FUNCTION Call_HMI

hmiHeaderInstance(NameApplication := 'Hochregallager',
				  OperatingModeHMIInterface := hmiOperatingmodeInterface,
				  HeaderHMIInterface := hmiHeaderInterface);
			  
hmiAdsCommunicationInterfaceInstance(Timeout := T#1S,
									 TimeoutHMI := T#500ms,
									 LocalAdsPort := 851,
									 HeartbeatHMI := hmiAdsCommunicationInterface.HeartbeatHMI);
									 

hmiAdsCommunicationInterface.DeviceIpAddress := hmiAdsCommunicationInterfaceInstance.LocalIpAddress;
hmiAdsCommunicationInterface.LocalAMSNetId := hmiAdsCommunicationInterfaceInstance.LocalAMSNetId;
hmiAdsCommunicationInterface.HeartbeatPLC := hmiAdsCommunicationInterfaceInstance.PLCHeartbeatHMICommunication;
hmiAdsCommunicationInterface.RuntimeStatus := hmiAdsCommunicationInterfaceInstance.AdsState;

END_FUNCTION

(* stored: Version 1.1.0.1
   POU Call_HMI: Id {619c281c-ef5d-4639-891a-10e7108f6cf6}, SpecialFunc None *)
